FUNCTION_BLOCK BufferedMoveToPosition IMPLEMENTS I_Task
VAR_INPUT
END_VAR
VAR_OUTPUT
END_VAR
VAR
	moveAbs : ARRAY[0..1] OF MoveAbs;
	iMoveAbs : I_MoveAbs := MoveAbs[0];
	moveAbsIndex : INT;
	_Axis : REFERENCE TO AXIS_REF;
	MoveToPosition : BOOL;
	State: INT;
	_Done: BOOL;
	_Error: BOOL;
	_Busy: BOOL;
END_VAR

{analysis -2}

METHOD Abort : BOOL
iMoveAbs.Execute := FALSE;
iMoveAbs.Position := 0;
iMoveAbs.Velocity := 0;
MoveToPosition := FALSE;
_Busy := FALSE;
Abort := TRUE;
State := 0;
END_METHOD

PROPERTY PUBLIC Acceleration : mc_lreal
GET
Acceleration := moveAbs[0].Acceleration;
END_GET
SET
MoveAbs[0].Acceleration := Acceleration;
MoveAbs[1].Acceleration := Acceleration;
END_SET
END_PROPERTY

PROPERTY BufferMode : MC_BufferMode
GET
BufferMode := MoveAbs[0].BufferMode;
END_GET
SET
MoveAbs[0].BufferMode := BufferMode;
MoveAbs[1].BufferMode := BufferMode;
END_SET
END_PROPERTY

PROPERTY Busy : BOOL
GET
Busy := _Busy;
END_GET
END_PROPERTY

METHOD Cycle : HRESULT
VAR_INPUT
END_VAR
Cycle := S_OK;
CASE State OF
	0:
		IF MoveToPosition THEN
			Cycle := S_PENDING;
			_Done := FALSE;
			_Error := FALSE;
			_Busy := TRUE;
			iMoveAbs.Execute := TRUE;
			IF iMoveAbs.Busy THEN
				State := 10;
				MoveToPosition := FALSE;
			END_IF
		END_IF
		
	10:
		IF NOT iMoveAbs.Busy THEN
			IF iMoveAbs.Done THEN
				_Done := TRUE;
			ELSIF iMoveAbs.Error THEN
				_Error := TRUE;
			END_IF
			_Busy := FALSE;
			iMoveAbs.Execute := FALSE;
			State := 0;
			Cycle := S_OK;
		END_IF
	ELSE
		Cycle := E_FAIL;
END_CASE

moveAbs[0](Axis := _Axis);
moveAbs[1](Axis := _Axis);
END_METHOD

PROPERTY PUBLIC Deceleration : mc_lreal
GET
Deceleration := MoveAbs[0].Deceleration;
END_GET
SET
MoveAbs[0].Deceleration := Deceleration;
MoveAbs[1].Deceleration := Deceleration;
END_SET
END_PROPERTY

PROPERTY Done : BOOL
GET
Done := _Done;
END_GET
END_PROPERTY

PROPERTY Error : BOOL
GET
Error := _Error;
END_GET
END_PROPERTY

METHOD FB_init : BOOL
VAR_INPUT
	bInitRetains : BOOL; // if TRUE, the retain variables are initialized (warm start / cold start)
	bInCopyCode : BOOL;  // if TRUE, the instance afterwards gets moved into the copy code (online change)
	axis : reference TO AXIS_REF;
END_VAR
_Axis REF= axis;
END_METHOD

PROPERTY PUBLIC Jerk : mc_lreal
GET
Jerk := MoveAbs[0].Jerk;
END_GET
SET
MoveAbs[0].Jerk := Jerk;
MoveAbs[1].Jerk := Jerk;
END_SET
END_PROPERTY

METHOD MoveTo : BOOL
VAR_INPUT
	Position : MC_LREAL;
	Velocity : MC_LREAL;
	Task : REFERENCE TO I_Task;
END_VAR
IF iMoveAbs.Execute THEN
	Abort();
	IF moveAbsIndex = 0 THEN
		moveAbsIndex := 1;
	ELSE
		moveAbsIndex := 0;
	END_IF
	iMoveAbs := moveAbs[moveAbsIndex];
END_IF

iMoveAbs.Position := Position;
iMoveAbs.Velocity := Velocity;
MoveToPosition := MoveTo := TRUE;
Task := THIS^;
END_METHOD

END_FUNCTION_BLOCK

(* stored: Version 1.1.0.1
   POU BufferedMoveToPosition: Id {f623c473-a640-4427-8dfd-9222a646d8bd}, SpecialFunc None
   Method Abort: Id {9045061b-9962-4607-8807-e07e05404656}
   Property Acceleration: Id {341f2499-163a-45c5-b240-f5c5cb02dff1}
   Get Get: Id {94f7a0b4-ef99-47e5-9f88-308be92cdbc4}
   Set Set: Id {dbd4bb19-bac7-45a6-9010-56d55b847137}
   Property BufferMode: Id {a7c0ed0c-36d3-453f-9975-ca4c3a7e9ba5}
   Get Get: Id {c282e09e-a818-4264-8f8d-0683a728c165}
   Set Set: Id {3591ccd7-2624-4277-b08d-05bb698ae34e}
   Property Busy: Id {1af2a4f9-8f2c-47f1-8f84-24d1cc3c56cc}
   Get Get: Id {d60afff3-b571-480e-8382-7cb6dec1c3d4}
   Method Cycle: Id {968b2426-4712-4973-a44f-8ea7571f0394}
   Property Deceleration: Id {15394e2a-7137-47ee-a0e9-ae4c783d030d}
   Get Get: Id {b409354e-6bdb-432b-bfed-d7faeda4d824}
   Set Set: Id {acdbbe46-8929-47eb-922e-1d284d954e8a}
   Property Done: Id {2efd6afe-2e1a-4877-9647-5bc5cdd99fbe}
   Get Get: Id {e37ef1fe-c5a1-4ddb-9b9d-cdaa750d2b2b}
   Property Error: Id {13f38694-36f8-4930-ab75-64619c3226f8}
   Get Get: Id {be92f53e-b6d5-425a-a3c4-51d3f85be2d7}
   Method FB_init: Id {06c8f2c4-26d3-46f9-a424-5aff24031530}
   Property Jerk: Id {c177883f-4564-4af8-a89b-8c0edf420990}
   Get Get: Id {5a0859c3-34f7-4dae-a686-377d861e0c51}
   Set Set: Id {6d085ea2-9832-4224-ada6-3f46c8535aed}
   Method MoveTo: Id {094fc655-ef28-4681-8db4-7d4b15208bc6} *)
